INTERFACE I_Tree_Map EXTENDS I_Map

// Traversal method for retrieving keys and values in the tree map set.
PROPERTY _Traversal : T_BST_Traversal
GET
END_GET
SET
END_SET
END_PROPERTY

END_INTERFACE

(* stored: Version 1.1.0.1
   Itf I_Tree_Map: Id {14451225-0556-0f35-2947-070bd85e3e19}
   Property _Traversal: Id {902f1fd8-d3e5-091f-1c7d-b6e0b9ae3e69}
   Get Get: Id {378a266b-aaf4-0962-14dd-47029a3e0ec3}
   Set Set: Id {04ff649f-7ba0-06a9-23d1-83bd539e1785} *)
